(* PLC project analog_sensor, Dassault Systèmes ControlBuild 2024x *)
(* stored: creationDateTime 2023-10-03T11:12:50-01:00 *)

(* This module simulates the behaviour of an analog sensor. It allows to create a fault on the measured quantity. *)
FUNCTION_BLOCK equipment_library.analog_sensor
  VAR_INPUT
    measure : REAL := 0.0;
    sensorSupply : BOOL := true;
  END_VAR
  VAR_OUTPUT
    realValue : REAL := 0.0;
    intValue : REAL := 0.0;
    dintValue : REAL := 0.0;
  END_VAR
  VAR
    tmp : DINT := 0;
    localValue : REAL := 0.0;
    nbDigit : SINT := 2;
  END_VAR
  VAR
    d_value : BOOL := false;
    v_d_value : REAL := 0.0;
  END_VAR


ACTION C_source_code:
/* ----------------------------------------------------------------	*/
/* Type : Model of Operative Behaviour					*/
/* Category :  Sensors							*/
/* Author : Dassault Systemes						*/
/* Update date : June 2018							*/
/* ----------------------------------------------------------------	*/
/* This module simulates the behaviour of an analog sensor.		*/
/* It allows to create a fault on the measured quantity. 		*/
/* ----------------------------------------------------------------	*/

if (d_value) localValue  = v_d_value;
else 
	if ( sensorSupply  ) localValue  = measure  ;
	else localValue   = 0.0;

/* On tronque la realValue d'affichage à 1,2,3,ou 4 digit derriere la virgule 	*/
if ((nbDigit > 4) || (nbDigit <= 0)) nbDigit = 2;
tmp = localValue  *  pow(10, nbDigit);
realValue = tmp / pow(10, nbDigit);

/* si le capteur depasse la plage autorisée, on force la valeur à 0 */
if ((realValue <= 32767) && (realValue >= -32768)) intValue = realValue;
	else intValue =0;

dintValue = realValue;
END_ACTION
END_FUNCTION_BLOCK
